TYPE DUT_ALM :
STRUCT
	IsHealthy: BOOL := TRUE;
	TimeFailure: BOOL := FALSE;
	InAlarm: BOOL := TimeFailure OR NOT (IsHealthy);
END_STRUCT
END_TYPE

(* stored: Version 1.1.0.1, ProductVersion 3.1.4024.12
   DUT DUT_ALM: Id {6758646b-b6b7-4d66-b478-11801b6873dc} *)
